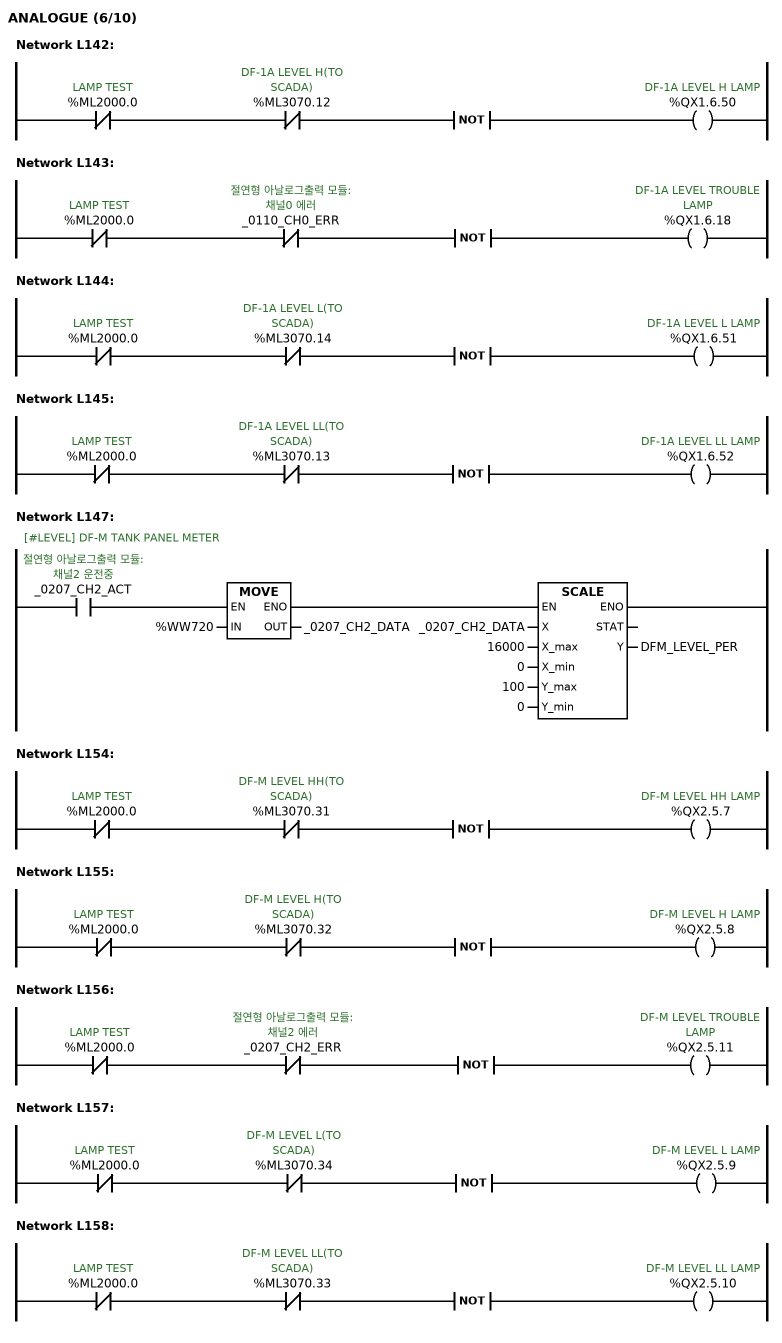
(* [picture p48: ANALOGUE rungs L142-L158] *)
(* Rung L142 *)
%QX1.6.50 := NOT (NOT %ML2000.0 AND NOT %ML3070.12);
(* Rung L143 *)
%QX1.6.18 := NOT (NOT %ML2000.0 AND NOT _0110_CH0_ERR);
(* Rung L144 *)
%QX1.6.51 := NOT (NOT %ML2000.0 AND NOT %ML3070.14);
(* Rung L145 *)
%QX1.6.52 := NOT (NOT %ML2000.0 AND NOT %ML3070.13);
(* [#LEVEL] DF-M TANK PANEL METER *)
(* Rung L147 *)
IF _0207_CH2_ACT THEN
    _0207_CH2_DATA := %WW720;
    SCALE(X := _0207_CH2_DATA, X_max := 16000, X_min := 0, Y_max := 100, Y_min := 0, Y => DFM_LEVEL_PER);
END_IF;
(* Rung L154 *)
%QX2.5.7 := NOT (NOT %ML2000.0 AND NOT %ML3070.31);
(* Rung L155 *)
%QX2.5.8 := NOT (NOT %ML2000.0 AND NOT %ML3070.32);
(* Rung L156 *)
%QX2.5.11 := NOT (NOT %ML2000.0 AND NOT _0207_CH2_ERR);
(* Rung L157 *)
%QX2.5.9 := NOT (NOT %ML2000.0 AND NOT %ML3070.34);
(* Rung L158 *)
%QX2.5.10 := NOT (NOT %ML2000.0 AND NOT %ML3070.33);

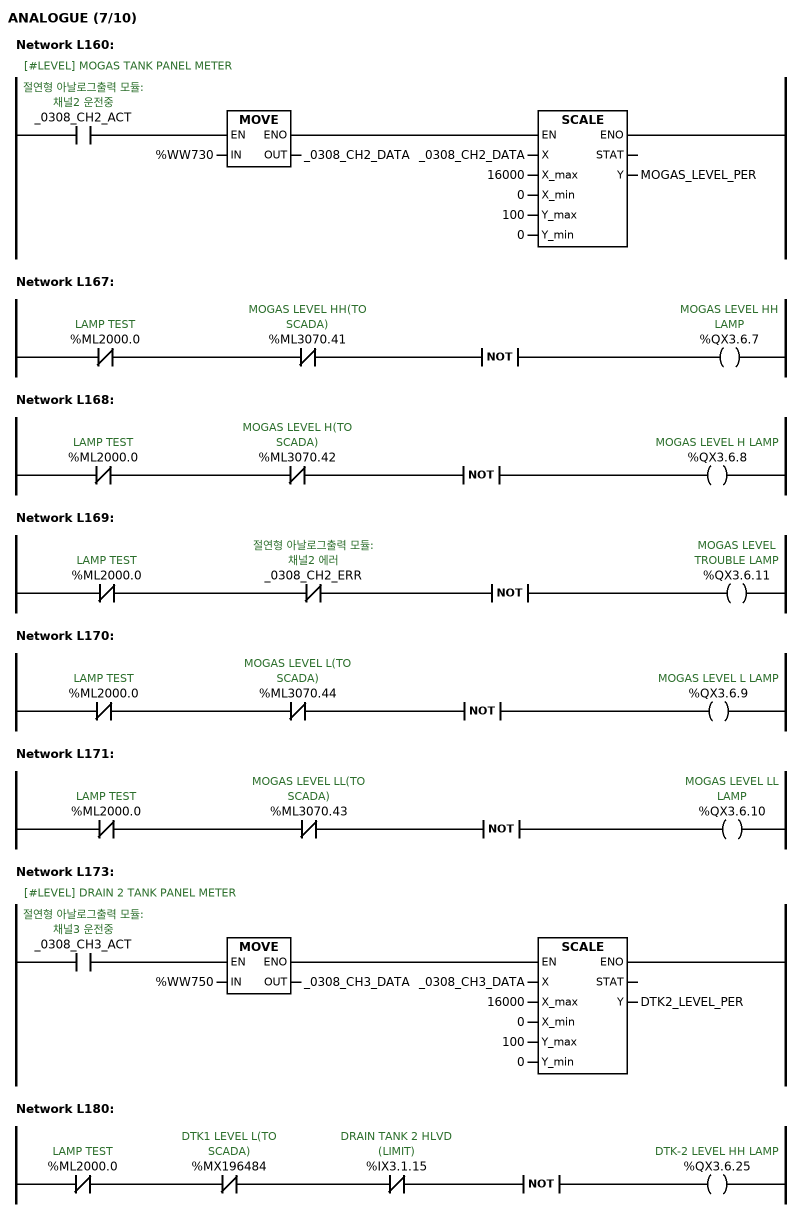
(* [#LEVEL] MOGAS TANK PANEL METER *)
(* Rung L160 *)
IF _0308_CH2_ACT THEN
    _0308_CH2_DATA := %WW730;
    SCALE(X := _0308_CH2_DATA, X_max := 16000, X_min := 0, Y_max := 100, Y_min := 0, Y => MOGAS_LEVEL_PER);
END_IF;
(* Rung L167 *)
%QX3.6.7 := NOT (NOT %ML2000.0 AND NOT %ML3070.41);
(* Rung L168 *)
%QX3.6.8 := NOT (NOT %ML2000.0 AND NOT %ML3070.42);
(* Rung L169 *)
%QX3.6.11 := NOT (NOT %ML2000.0 AND NOT _0308_CH2_ERR);
(* Rung L170 *)
%QX3.6.9 := NOT (NOT %ML2000.0 AND NOT %ML3070.44);
(* Rung L171 *)
%QX3.6.10 := NOT (NOT %ML2000.0 AND NOT %ML3070.43);
(* [#LEVEL] DRAIN 2 TANK PANEL METER *)
(* Rung L173 *)
IF _0308_CH3_ACT THEN
    _0308_CH3_DATA := %WW750;
    SCALE(X := _0308_CH3_DATA, X_max := 16000, X_min := 0, Y_max := 100, Y_min := 0, Y => DTK2_LEVEL_PER);
END_IF;
(* Rung L180 *)
%QX3.6.25 := NOT (NOT %ML2000.0 AND NOT %MX196484 AND NOT %IX3.1.15);

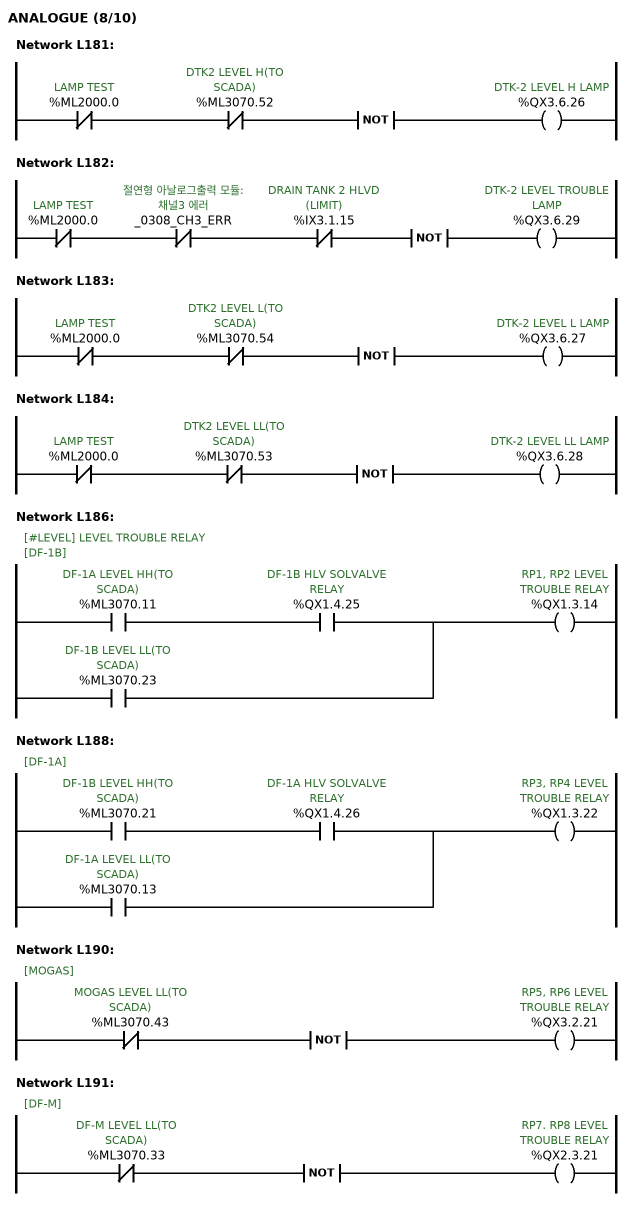
(* Rung L181 *)
%QX3.6.26 := NOT (NOT %ML2000.0 AND NOT %ML3070.52);
(* Rung L182 *)
%QX3.6.29 := NOT (NOT %ML2000.0 AND NOT _0308_CH3_ERR AND NOT %IX3.1.15);
(* Rung L183 *)
%QX3.6.27 := NOT (NOT %ML2000.0 AND NOT %ML3070.54);
(* Rung L184 *)
%QX3.6.28 := NOT (NOT %ML2000.0 AND NOT %ML3070.53);
(* [#LEVEL] LEVEL TROUBLE RELAY *)
(* Rung L186 *)
%QX1.3.14 := (%ML3070.11 AND %QX1.4.25) OR %ML3070.23;
(* [DF-1B] *)
(* Rung L188 *)
%QX1.3.22 := (%ML3070.21 AND %QX1.4.26) OR %ML3070.13;
(* [DF-1A] *)
(* Rung L190 *)
%QX3.2.21 := %ML3070.43;
(* [MOGAS] *)
(* Rung L191 *)
%QX2.3.21 := %ML3070.33;
(* [DF-M] *)

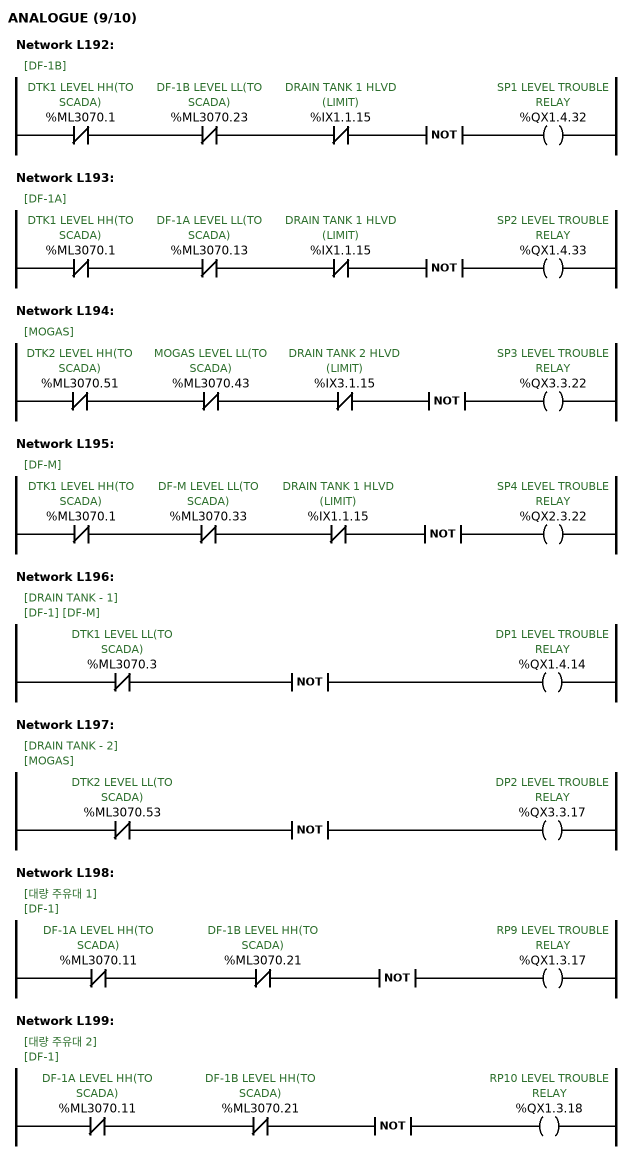
(* Rung L192 *)
%QX1.4.32 := NOT (NOT %ML3070.1 AND NOT %ML3070.23 AND NOT %IX1.1.15);
(* [DF-1B] *)
(* Rung L193 *)
%QX1.4.33 := NOT (NOT %ML3070.1 AND NOT %ML3070.13 AND NOT %IX1.1.15);
(* [DF-1A] *)
(* Rung L194 *)
%QX3.3.22 := NOT (NOT %ML3070.51 AND NOT %ML3070.43 AND NOT %IX3.1.15);
(* [MOGAS] *)
(* Rung L195 *)
%QX2.3.22 := NOT (NOT %ML3070.1 AND NOT %ML3070.33 AND NOT %IX1.1.15);
(* [DF-M] *)
(* Rung L196 *)
%QX1.4.14 := %ML3070.3;
(* [DRAIN TANK - 1] / [DF-1] [DF-M] *)
(* Rung L197 *)
%QX3.3.17 := %ML3070.53;
(* [DRAIN TANK - 2] / [MOGAS] *)
(* Rung L198 *)
%QX1.3.17 := NOT (NOT %ML3070.11 AND NOT %ML3070.21);
(* [대량 주유대 1] / [DF-1] *)
(* Rung L199 *)
%QX1.3.18 := NOT (NOT %ML3070.11 AND NOT %ML3070.21);
(* [대량 주유대 2] / [DF-1] *)

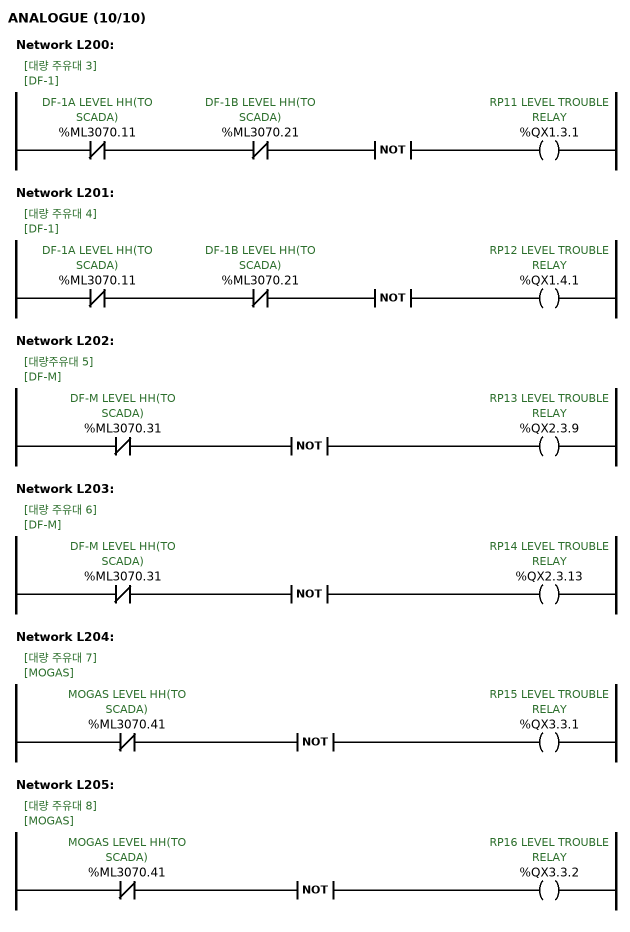
(* Rung L200 *)
%QX1.3.1 := NOT (NOT %ML3070.11 AND NOT %ML3070.21);
(* [대량 주유대 3] / [DF-1] *)
(* Rung L201 *)
%QX1.4.1 := NOT (NOT %ML3070.11 AND NOT %ML3070.21);
(* [대량 주유대 4] / [DF-1] *)
(* Rung L202 *)
%QX2.3.9 := %ML3070.31;
(* [대량주유대 5] / [DF-M] *)
(* Rung L203 *)
%QX2.3.13 := %ML3070.31;
(* [대량 주유대 6] / [DF-M] *)
(* Rung L204 *)
%QX3.3.1 := %ML3070.41;
(* [대량 주유대 7] / [MOGAS] *)
(* Rung L205 *)
%QX3.3.2 := %ML3070.41;
(* [대량 주유대 8] / [MOGAS] *)
END_PROGRAM

PROGRAM COMMUNICATION (* task: 스캔 프로그램 *)

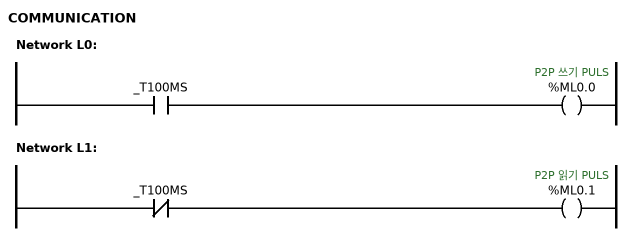
(* Rung L0 *)
%ML0.0 := _T100MS;
(* Rung L1 *)
%ML0.1 := NOT _T100MS;
END_PROGRAM

PROGRAM SCADA (* task: 스캔 프로그램 *)
VAR
    DFM_anyRun_SW : BOOL;
    MOGAS_anyRun_SW : BOOL;
END_VAR
VAR
    _t1 : BOOL;
    _t2 : BOOL;
END_VAR

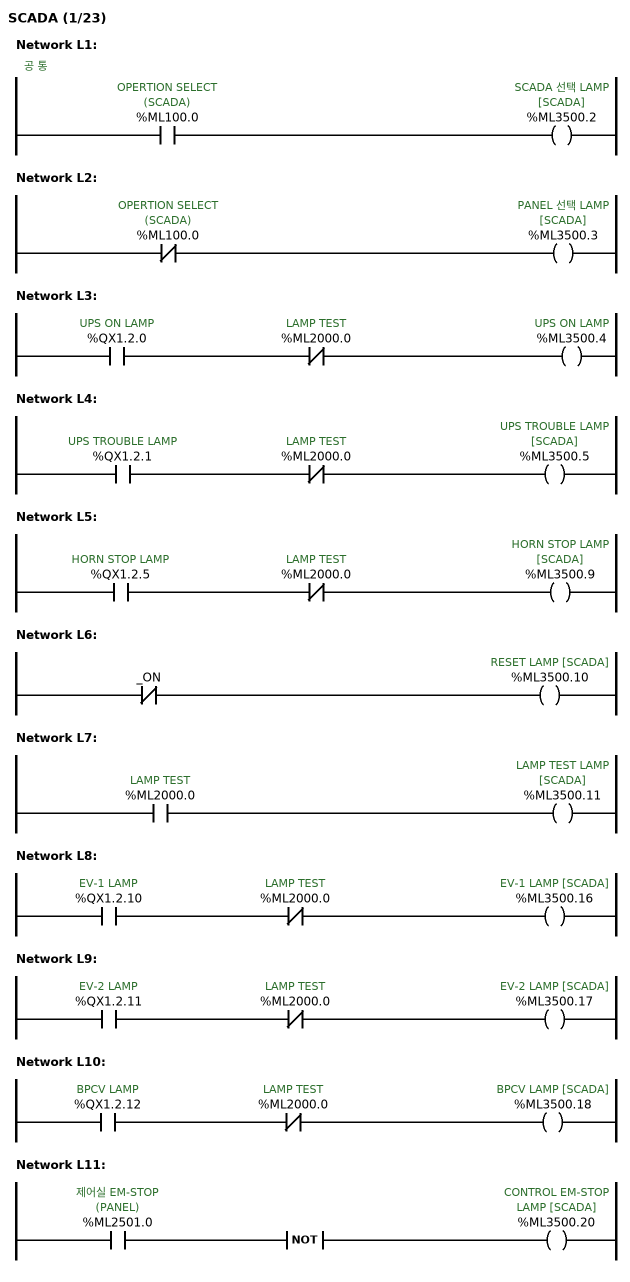
(* 공 통 *)
(* Rung L1 *)
%ML3500.2 := %ML100.0;
(* Rung L2 *)
%ML3500.3 := NOT %ML100.0;
(* Rung L3 *)
%ML3500.4 := %QX1.2.0 AND NOT %ML2000.0;
(* Rung L4 *)
%ML3500.5 := %QX1.2.1 AND NOT %ML2000.0;
(* Rung L5 *)
%ML3500.9 := %QX1.2.5 AND NOT %ML2000.0;
(* Rung L6 *)
%ML3500.10 := NOT _ON;
(* Rung L7 *)
%ML3500.11 := %ML2000.0;
(* Rung L8 *)
%ML3500.16 := %QX1.2.10 AND NOT %ML2000.0;
(* Rung L9 *)
%ML3500.17 := %QX1.2.11 AND NOT %ML2000.0;
(* Rung L10 *)
%ML3500.18 := %QX1.2.12 AND NOT %ML2000.0;
(* Rung L11 *)
%ML3500.20 := NOT %ML2501.0;

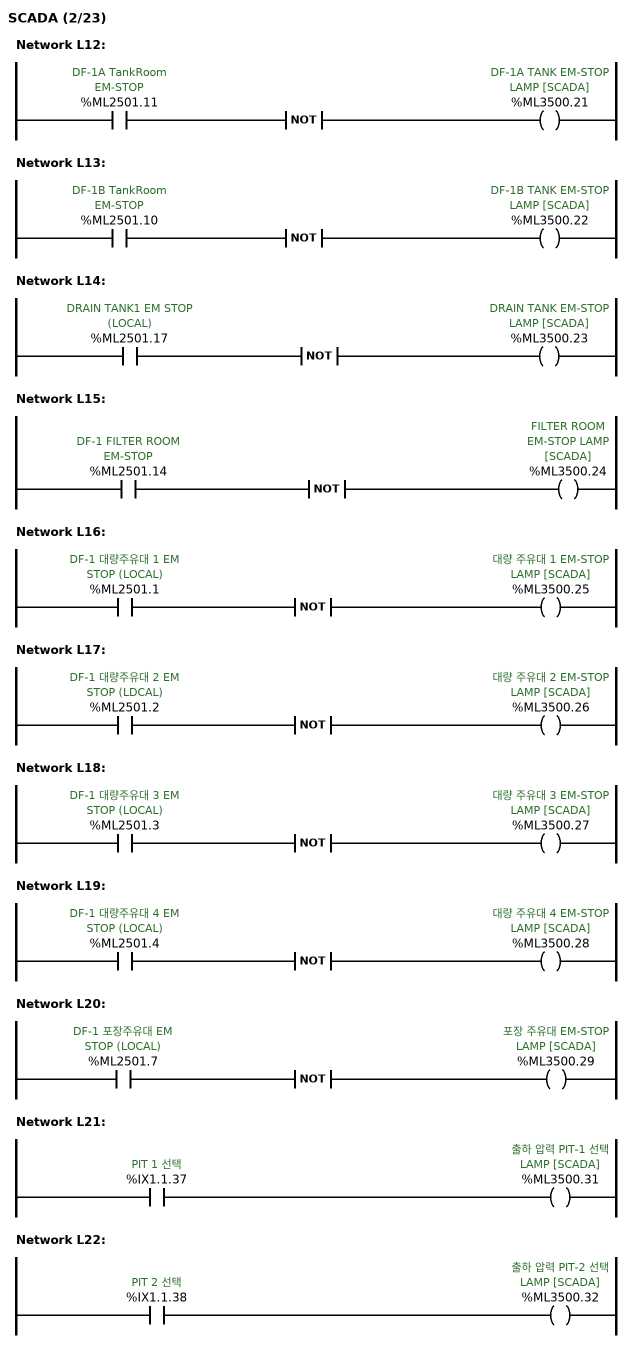
(* Rung L12 *)
%ML3500.21 := NOT %ML2501.11;
(* Rung L13 *)
%ML3500.22 := NOT %ML2501.10;
(* Rung L14 *)
%ML3500.23 := NOT %ML2501.17;
(* Rung L15 *)
%ML3500.24 := NOT %ML2501.14;
(* Rung L16 *)
%ML3500.25 := NOT %ML2501.1;
(* Rung L17 *)
%ML3500.26 := NOT %ML2501.2;
(* Rung L18 *)
%ML3500.27 := NOT %ML2501.3;
(* Rung L19 *)
%ML3500.28 := NOT %ML2501.4;
(* Rung L20 *)
%ML3500.29 := NOT %ML2501.7;
(* Rung L21 *)
%ML3500.31 := %IX1.1.37;
(* Rung L22 *)
%ML3500.32 := %IX1.1.38;

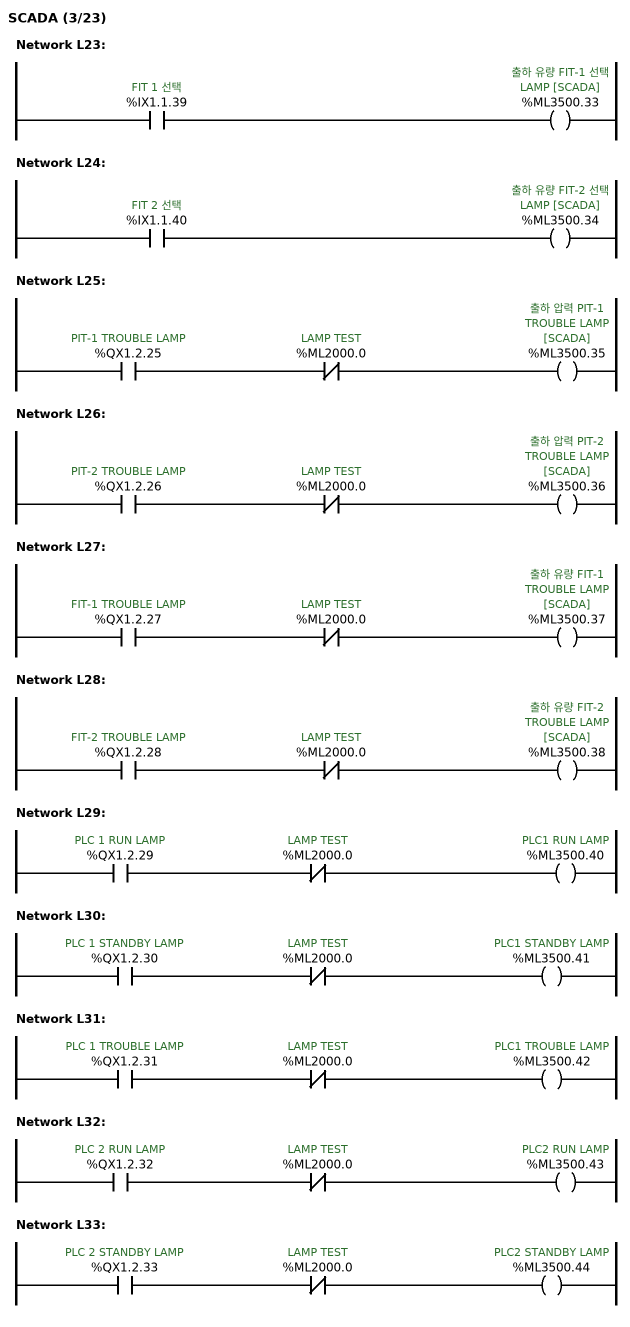
(* Rung L23 *)
%ML3500.33 := %IX1.1.39;
(* Rung L24 *)
%ML3500.34 := %IX1.1.40;
(* Rung L25 *)
%ML3500.35 := %QX1.2.25 AND NOT %ML2000.0;
(* Rung L26 *)
%ML3500.36 := %QX1.2.26 AND NOT %ML2000.0;
(* Rung L27 *)
%ML3500.37 := %QX1.2.27 AND NOT %ML2000.0;
(* Rung L28 *)
%ML3500.38 := %QX1.2.28 AND NOT %ML2000.0;
(* Rung L29 *)
%ML3500.40 := %QX1.2.29 AND NOT %ML2000.0;
(* Rung L30 *)
%ML3500.41 := %QX1.2.30 AND NOT %ML2000.0;
(* Rung L31 *)
%ML3500.42 := %QX1.2.31 AND NOT %ML2000.0;
(* Rung L32 *)
%ML3500.43 := %QX1.2.32 AND NOT %ML2000.0;
(* Rung L33 *)
%ML3500.44 := %QX1.2.33 AND NOT %ML2000.0;

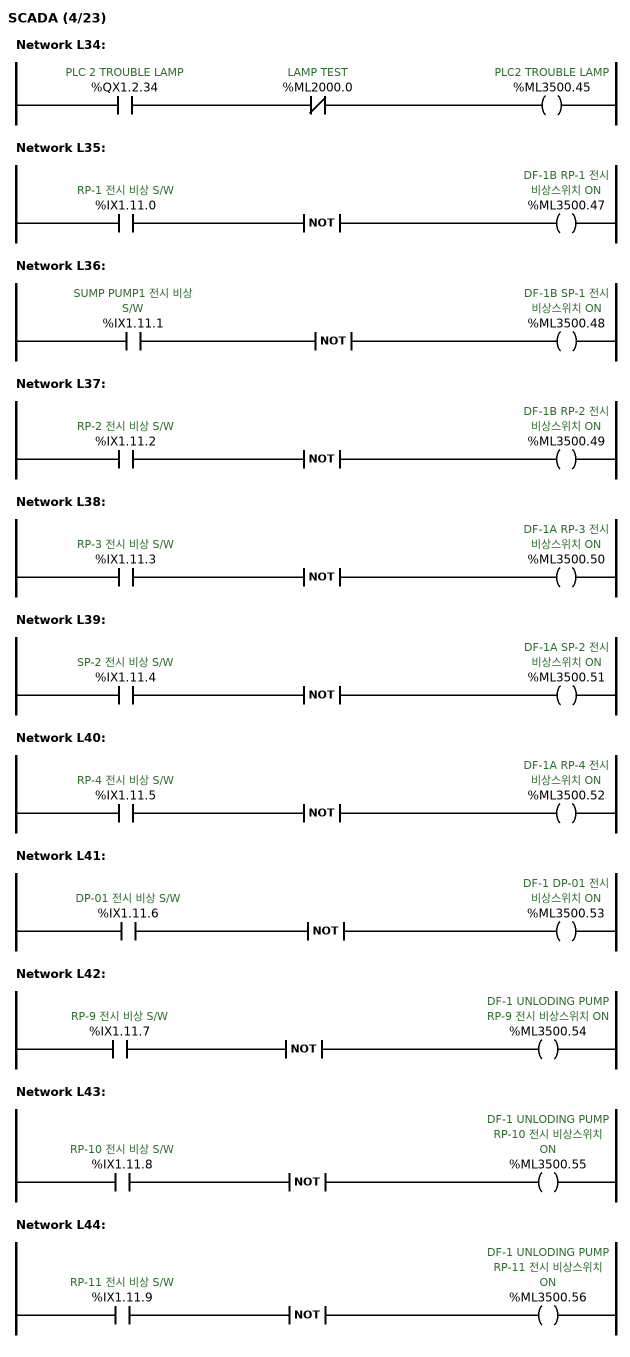
(* Rung L34 *)
%ML3500.45 := %QX1.2.34 AND NOT %ML2000.0;
(* Rung L35 *)
%ML3500.47 := NOT %IX1.11.0;
(* Rung L36 *)
%ML3500.48 := NOT %IX1.11.1;
(* Rung L37 *)
%ML3500.49 := NOT %IX1.11.2;
(* Rung L38 *)
%ML3500.50 := NOT %IX1.11.3;
(* Rung L39 *)
%ML3500.51 := NOT %IX1.11.4;
(* Rung L40 *)
%ML3500.52 := NOT %IX1.11.5;
(* Rung L41 *)
%ML3500.53 := NOT %IX1.11.6;
(* Rung L42 *)
%ML3500.54 := NOT %IX1.11.7;
(* Rung L43 *)
%ML3500.55 := NOT %IX1.11.8;
(* Rung L44 *)
%ML3500.56 := NOT %IX1.11.9;

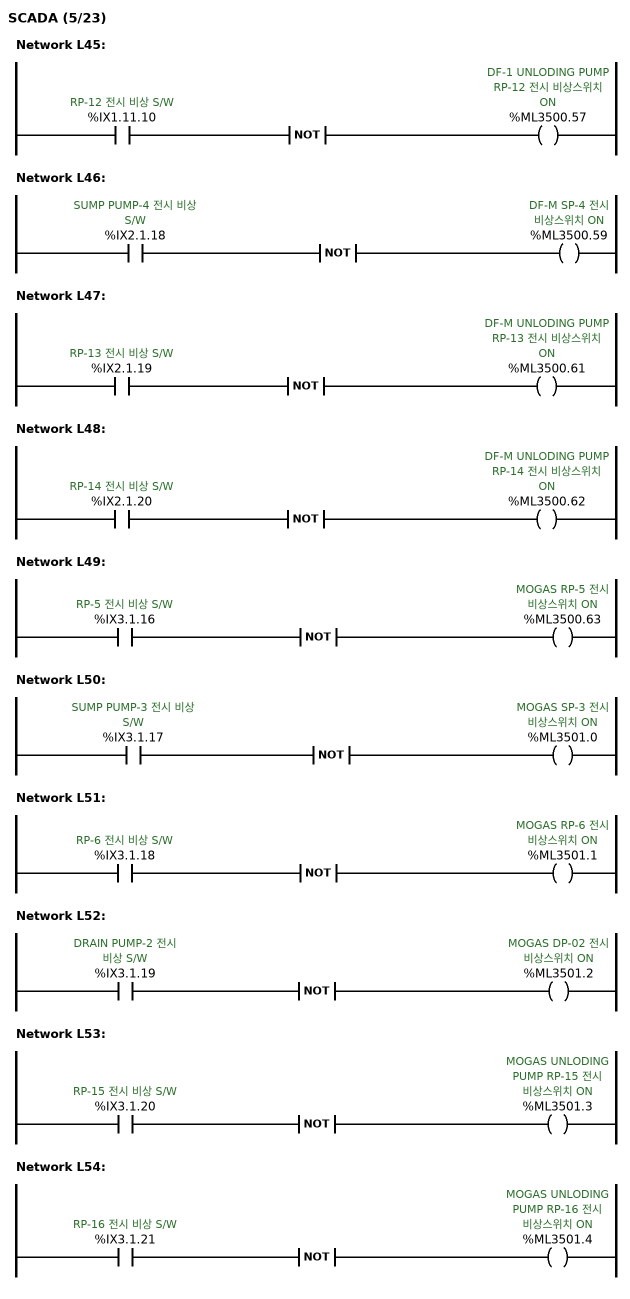
(* Rung L45 *)
%ML3500.57 := NOT %IX1.11.10;
(* Rung L46 *)
%ML3500.59 := NOT %IX2.1.18;
(* Rung L47 *)
%ML3500.61 := NOT %IX2.1.19;
(* Rung L48 *)
%ML3500.62 := NOT %IX2.1.20;
(* Rung L49 *)
%ML3500.63 := NOT %IX3.1.16;
(* Rung L50 *)
%ML3501.0 := NOT %IX3.1.17;
(* Rung L51 *)
%ML3501.1 := NOT %IX3.1.18;
(* Rung L52 *)
%ML3501.2 := NOT %IX3.1.19;
(* Rung L53 *)
%ML3501.3 := NOT %IX3.1.20;
(* Rung L54 *)
%ML3501.4 := NOT %IX3.1.21;

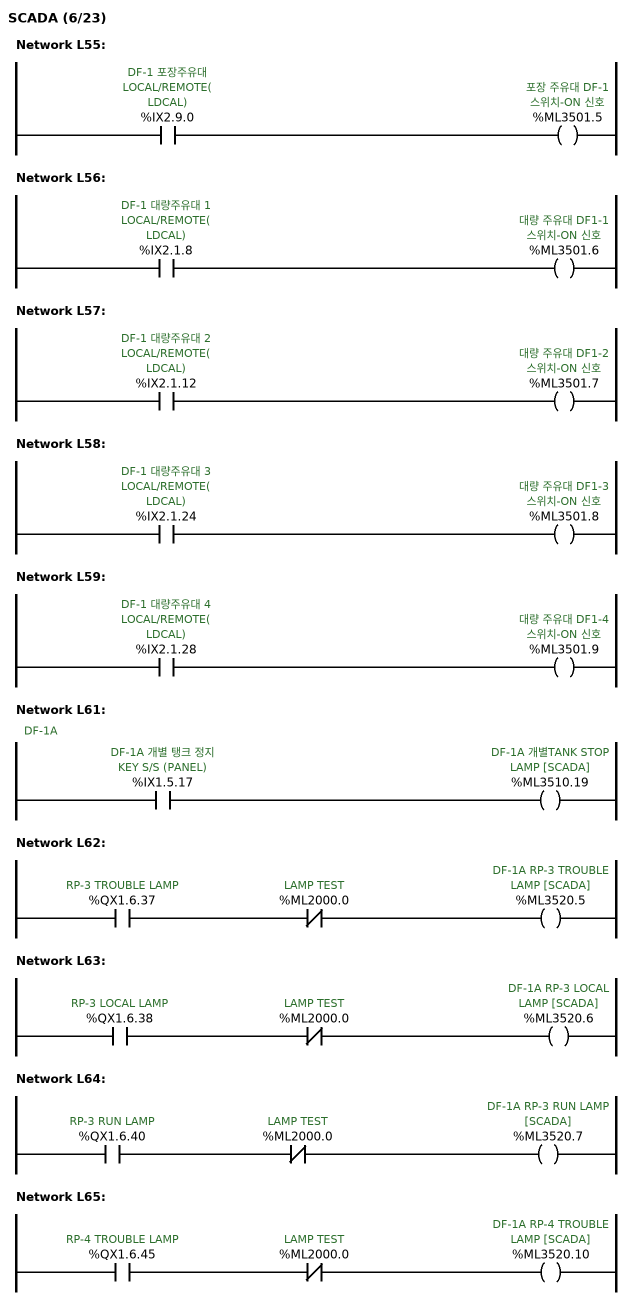
(* Rung L55 *)
%ML3501.5 := %IX2.9.0;
(* Rung L56 *)
%ML3501.6 := %IX2.1.8;
(* Rung L57 *)
%ML3501.7 := %IX2.1.12;
(* Rung L58 *)
%ML3501.8 := %IX2.1.24;
(* Rung L59 *)
%ML3501.9 := %IX2.1.28;
(* DF-1A *)
(* Rung L61 *)
%ML3510.19 := %IX1.5.17;
(* Rung L62 *)
%ML3520.5 := %QX1.6.37 AND NOT %ML2000.0;
(* Rung L63 *)
%ML3520.6 := %QX1.6.38 AND NOT %ML2000.0;
(* Rung L64 *)
%ML3520.7 := %QX1.6.40 AND NOT %ML2000.0;
(* Rung L65 *)
%ML3520.10 := %QX1.6.45 AND NOT %ML2000.0;

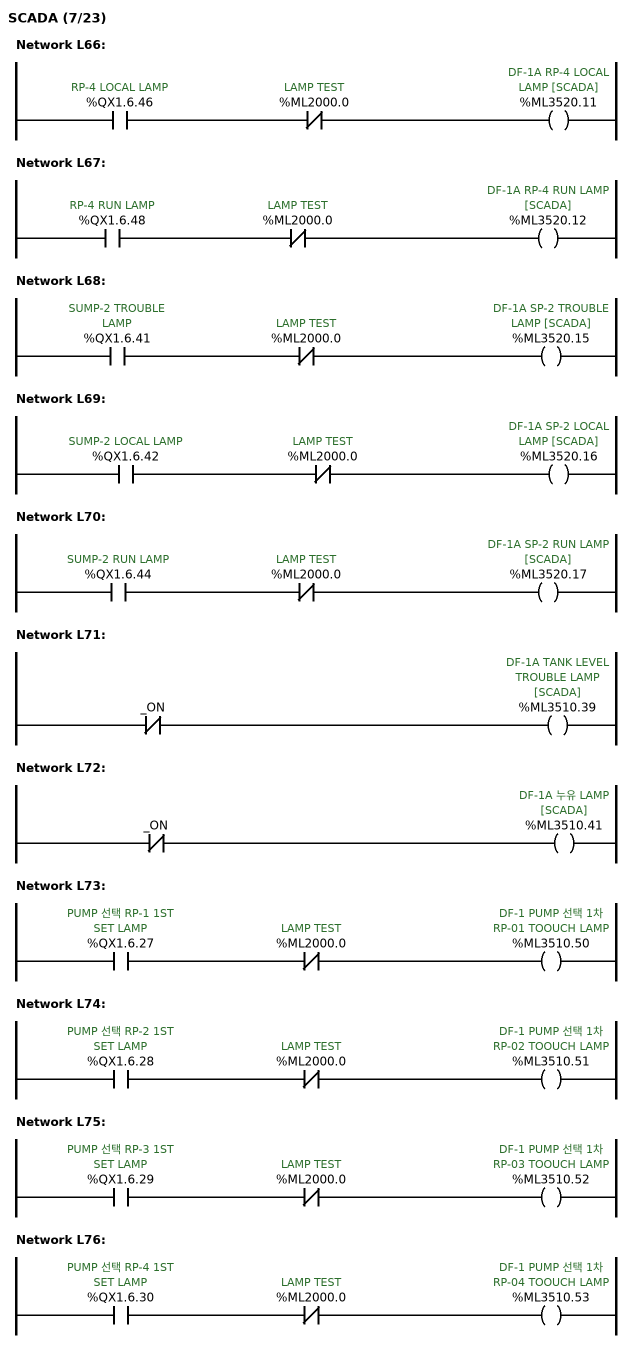
(* Rung L66 *)
%ML3520.11 := %QX1.6.46 AND NOT %ML2000.0;
(* Rung L67 *)
%ML3520.12 := %QX1.6.48 AND NOT %ML2000.0;
(* Rung L68 *)
%ML3520.15 := %QX1.6.41 AND NOT %ML2000.0;
(* Rung L69 *)
%ML3520.16 := %QX1.6.42 AND NOT %ML2000.0;
(* Rung L70 *)
%ML3520.17 := %QX1.6.44 AND NOT %ML2000.0;
(* Rung L71 *)
%ML3510.39 := NOT _ON;
(* Rung L72 *)
%ML3510.41 := NOT _ON;
(* Rung L73 *)
%ML3510.50 := %QX1.6.27 AND NOT %ML2000.0;
(* Rung L74 *)
%ML3510.51 := %QX1.6.28 AND NOT %ML2000.0;
(* Rung L75 *)
%ML3510.52 := %QX1.6.29 AND NOT %ML2000.0;
(* Rung L76 *)
%ML3510.53 := %QX1.6.30 AND NOT %ML2000.0;

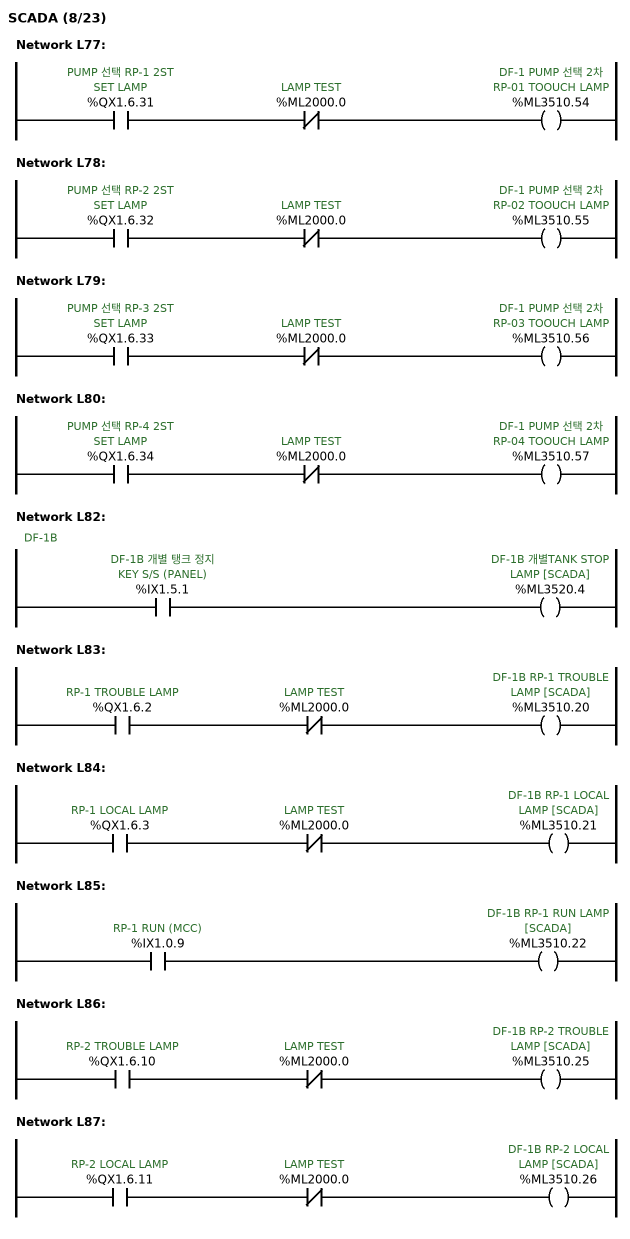
(* Rung L77 *)
%ML3510.54 := %QX1.6.31 AND NOT %ML2000.0;
(* Rung L78 *)
%ML3510.55 := %QX1.6.32 AND NOT %ML2000.0;
(* Rung L79 *)
%ML3510.56 := %QX1.6.33 AND NOT %ML2000.0;
(* Rung L80 *)
%ML3510.57 := %QX1.6.34 AND NOT %ML2000.0;
(* DF-1B *)
(* Rung L82 *)
%ML3520.4 := %IX1.5.1;
(* Rung L83 *)
%ML3510.20 := %QX1.6.2 AND NOT %ML2000.0;
(* Rung L84 *)
%ML3510.21 := %QX1.6.3 AND NOT %ML2000.0;
(* Rung L85 *)
%ML3510.22 := %IX1.0.9;
(* Rung L86 *)
%ML3510.25 := %QX1.6.10 AND NOT %ML2000.0;
(* Rung L87 *)
%ML3510.26 := %QX1.6.11 AND NOT %ML2000.0;

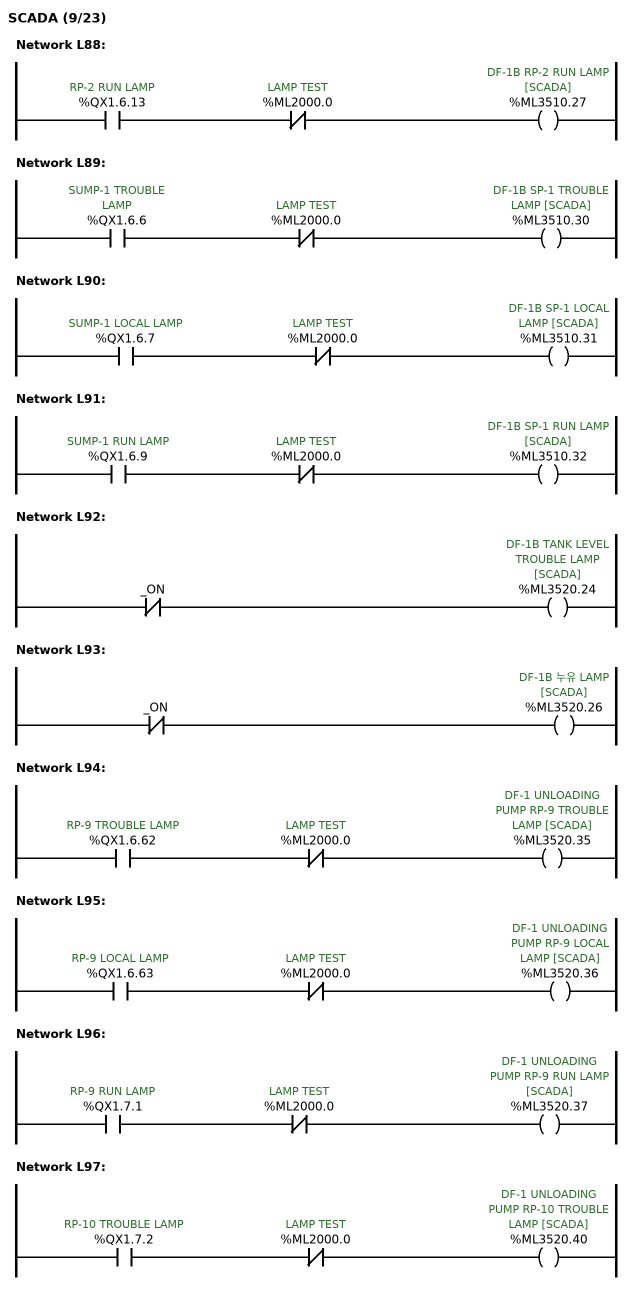
(* Rung L88 *)
%ML3510.27 := %QX1.6.13 AND NOT %ML2000.0;
(* Rung L89 *)
%ML3510.30 := %QX1.6.6 AND NOT %ML2000.0;
(* Rung L90 *)
%ML3510.31 := %QX1.6.7 AND NOT %ML2000.0;
(* Rung L91 *)
%ML3510.32 := %QX1.6.9 AND NOT %ML2000.0;
(* Rung L92 *)
%ML3520.24 := NOT _ON;
(* Rung L93 *)
%ML3520.26 := NOT _ON;
(* Rung L94 *)
%ML3520.35 := %QX1.6.62 AND NOT %ML2000.0;
(* Rung L95 *)
%ML3520.36 := %QX1.6.63 AND NOT %ML2000.0;
(* Rung L96 *)
%ML3520.37 := %QX1.7.1 AND NOT %ML2000.0;
(* Rung L97 *)
%ML3520.40 := %QX1.7.2 AND NOT %ML2000.0;

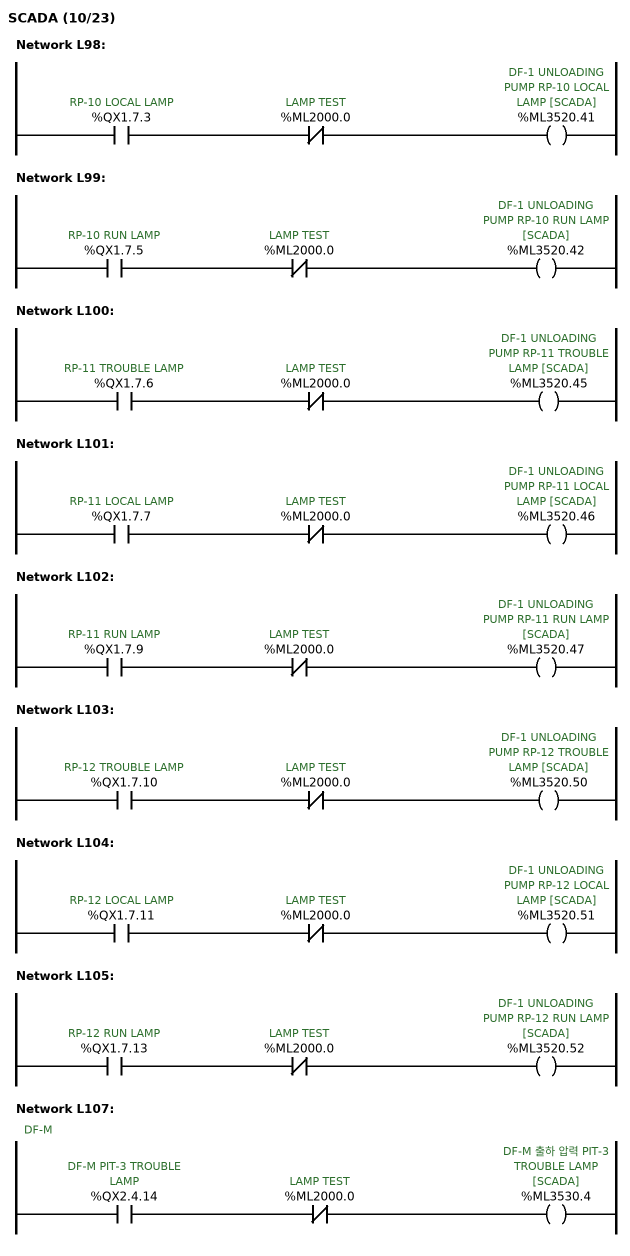
(* Rung L98 *)
%ML3520.41 := %QX1.7.3 AND NOT %ML2000.0;
(* Rung L99 *)
%ML3520.42 := %QX1.7.5 AND NOT %ML2000.0;
(* Rung L100 *)
%ML3520.45 := %QX1.7.6 AND NOT %ML2000.0;
(* Rung L101 *)
%ML3520.46 := %QX1.7.7 AND NOT %ML2000.0;
(* Rung L102 *)
%ML3520.47 := %QX1.7.9 AND NOT %ML2000.0;
(* Rung L103 *)
%ML3520.50 := %QX1.7.10 AND NOT %ML2000.0;
(* Rung L104 *)
%ML3520.51 := %QX1.7.11 AND NOT %ML2000.0;
(* Rung L105 *)
%ML3520.52 := %QX1.7.13 AND NOT %ML2000.0;
(* DF-M *)
(* Rung L107 *)
%ML3530.4 := %QX2.4.14 AND NOT %ML2000.0;

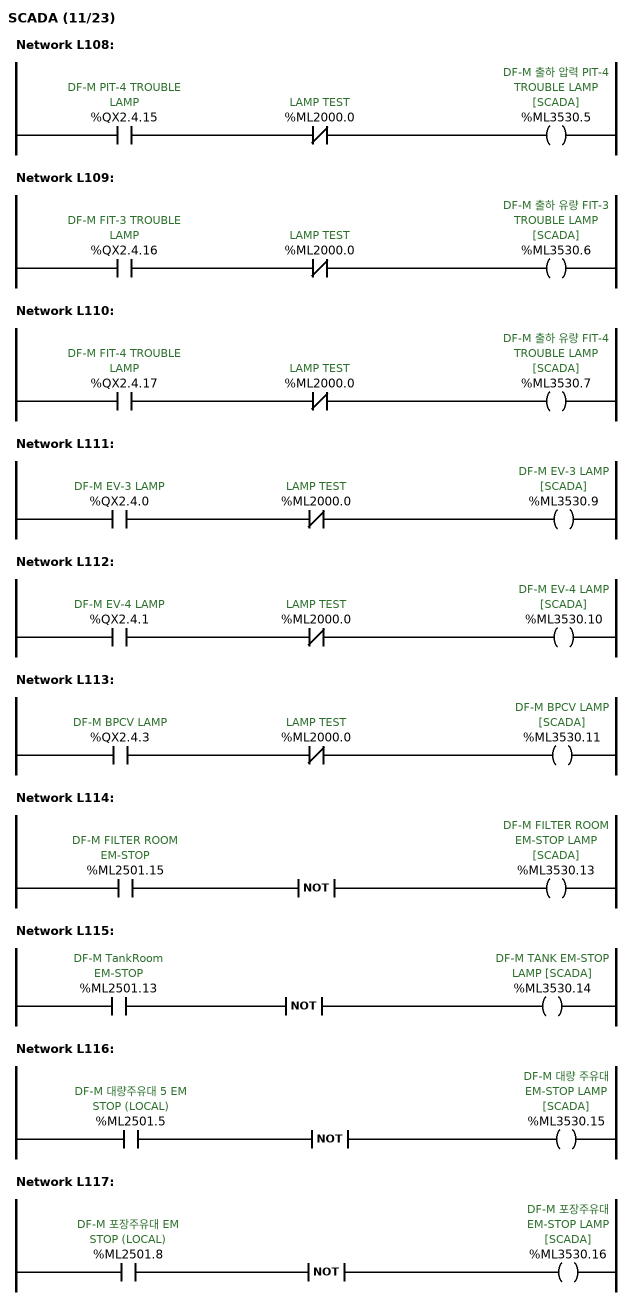
(* Rung L108 *)
%ML3530.5 := %QX2.4.15 AND NOT %ML2000.0;
(* Rung L109 *)
%ML3530.6 := %QX2.4.16 AND NOT %ML2000.0;
(* Rung L110 *)
%ML3530.7 := %QX2.4.17 AND NOT %ML2000.0;
(* Rung L111 *)
%ML3530.9 := %QX2.4.0 AND NOT %ML2000.0;
(* Rung L112 *)
%ML3530.10 := %QX2.4.1 AND NOT %ML2000.0;
(* Rung L113 *)
%ML3530.11 := %QX2.4.3 AND NOT %ML2000.0;
(* Rung L114 *)
%ML3530.13 := NOT %ML2501.15;
(* Rung L115 *)
%ML3530.14 := NOT %ML2501.13;
(* Rung L116 *)
%ML3530.15 := NOT %ML2501.5;
(* Rung L117 *)
%ML3530.16 := NOT %ML2501.8;

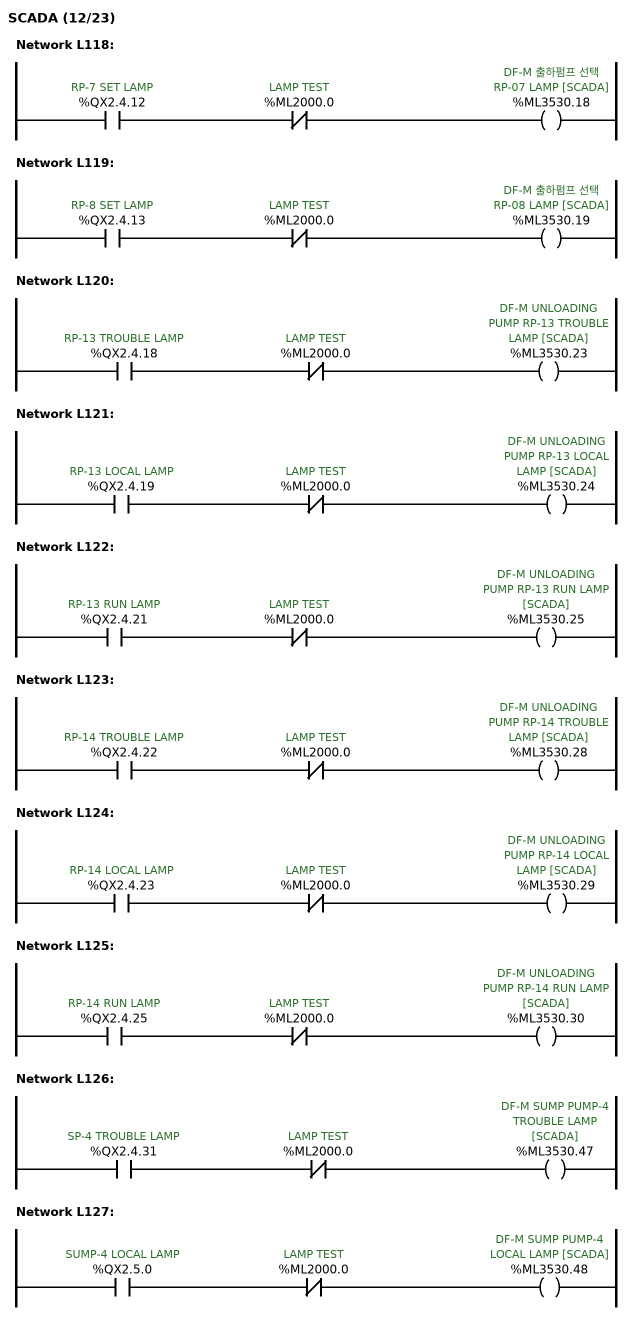
(* Rung L118 *)
%ML3530.18 := %QX2.4.12 AND NOT %ML2000.0;
(* Rung L119 *)
%ML3530.19 := %QX2.4.13 AND NOT %ML2000.0;
(* Rung L120 *)
%ML3530.23 := %QX2.4.18 AND NOT %ML2000.0;
(* Rung L121 *)
%ML3530.24 := %QX2.4.19 AND NOT %ML2000.0;
(* Rung L122 *)
%ML3530.25 := %QX2.4.21 AND NOT %ML2000.0;
(* Rung L123 *)
%ML3530.28 := %QX2.4.22 AND NOT %ML2000.0;
(* Rung L124 *)
%ML3530.29 := %QX2.4.23 AND NOT %ML2000.0;
(* Rung L125 *)
%ML3530.30 := %QX2.4.25 AND NOT %ML2000.0;
(* Rung L126 *)
%ML3530.47 := %QX2.4.31 AND NOT %ML2000.0;
(* Rung L127 *)
%ML3530.48 := %QX2.5.0 AND NOT %ML2000.0;

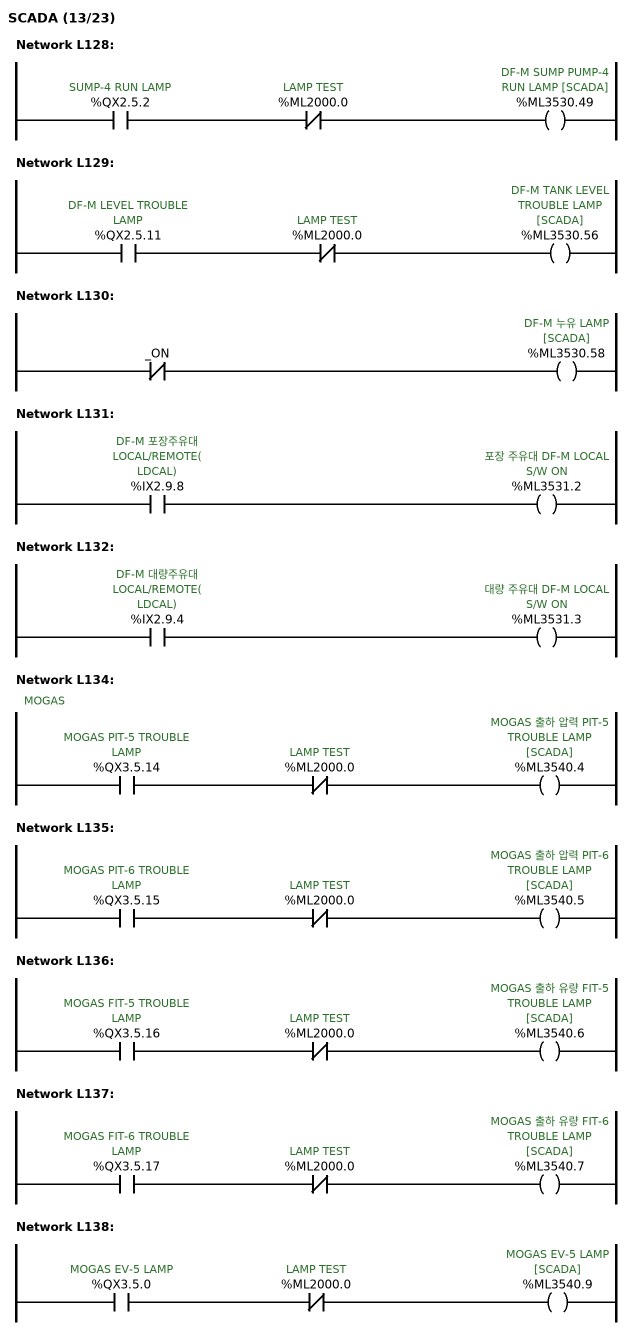
(* Rung L128 *)
%ML3530.49 := %QX2.5.2 AND NOT %ML2000.0;
(* Rung L129 *)
%ML3530.56 := %QX2.5.11 AND NOT %ML2000.0;
(* Rung L130 *)
%ML3530.58 := NOT _ON;
(* Rung L131 *)
%ML3531.2 := %IX2.9.8;
(* Rung L132 *)
%ML3531.3 := %IX2.9.4;
(* MOGAS *)
(* Rung L134 *)
%ML3540.4 := %QX3.5.14 AND NOT %ML2000.0;
(* Rung L135 *)
%ML3540.5 := %QX3.5.15 AND NOT %ML2000.0;
(* Rung L136 *)
%ML3540.6 := %QX3.5.16 AND NOT %ML2000.0;
(* Rung L137 *)
%ML3540.7 := %QX3.5.17 AND NOT %ML2000.0;
(* Rung L138 *)
%ML3540.9 := %QX3.5.0 AND NOT %ML2000.0;

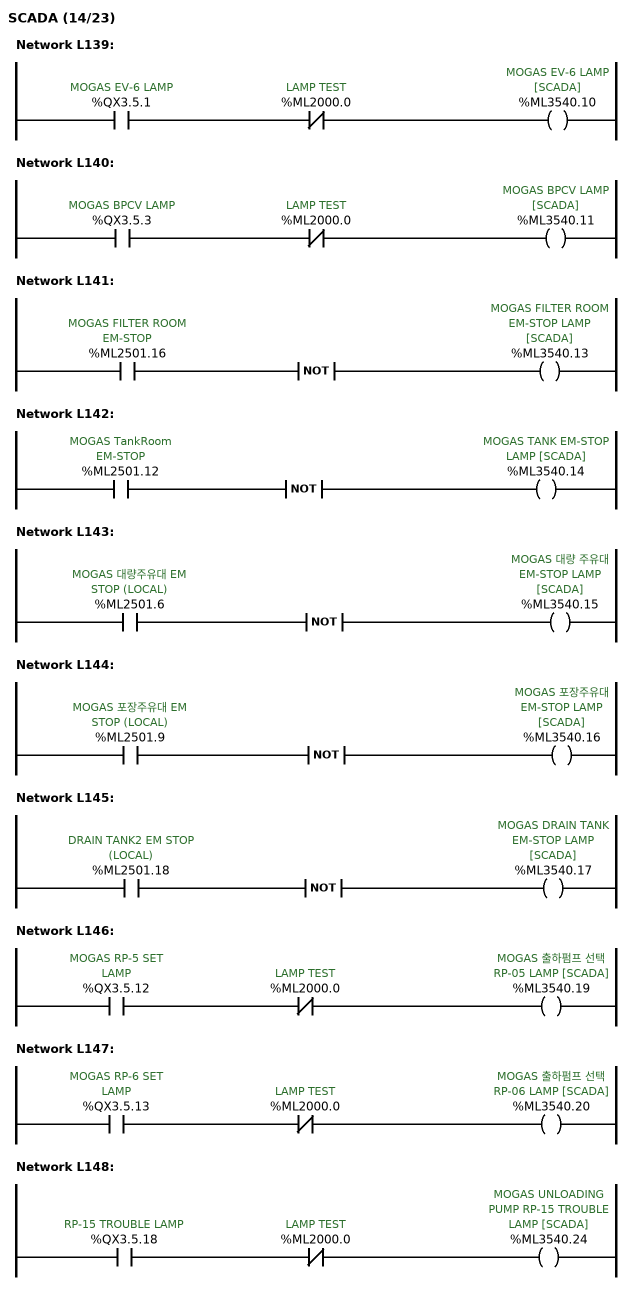
(* Rung L139 *)
%ML3540.10 := %QX3.5.1 AND NOT %ML2000.0;
(* Rung L140 *)
%ML3540.11 := %QX3.5.3 AND NOT %ML2000.0;
(* Rung L141 *)
%ML3540.13 := NOT %ML2501.16;
(* Rung L142 *)
%ML3540.14 := NOT %ML2501.12;
(* Rung L143 *)
%ML3540.15 := NOT %ML2501.6;
(* Rung L144 *)
%ML3540.16 := NOT %ML2501.9;
(* Rung L145 *)
%ML3540.17 := NOT %ML2501.18;
(* Rung L146 *)
%ML3540.19 := %QX3.5.12 AND NOT %ML2000.0;
(* Rung L147 *)
%ML3540.20 := %QX3.5.13 AND NOT %ML2000.0;
(* Rung L148 *)
%ML3540.24 := %QX3.5.18 AND NOT %ML2000.0;

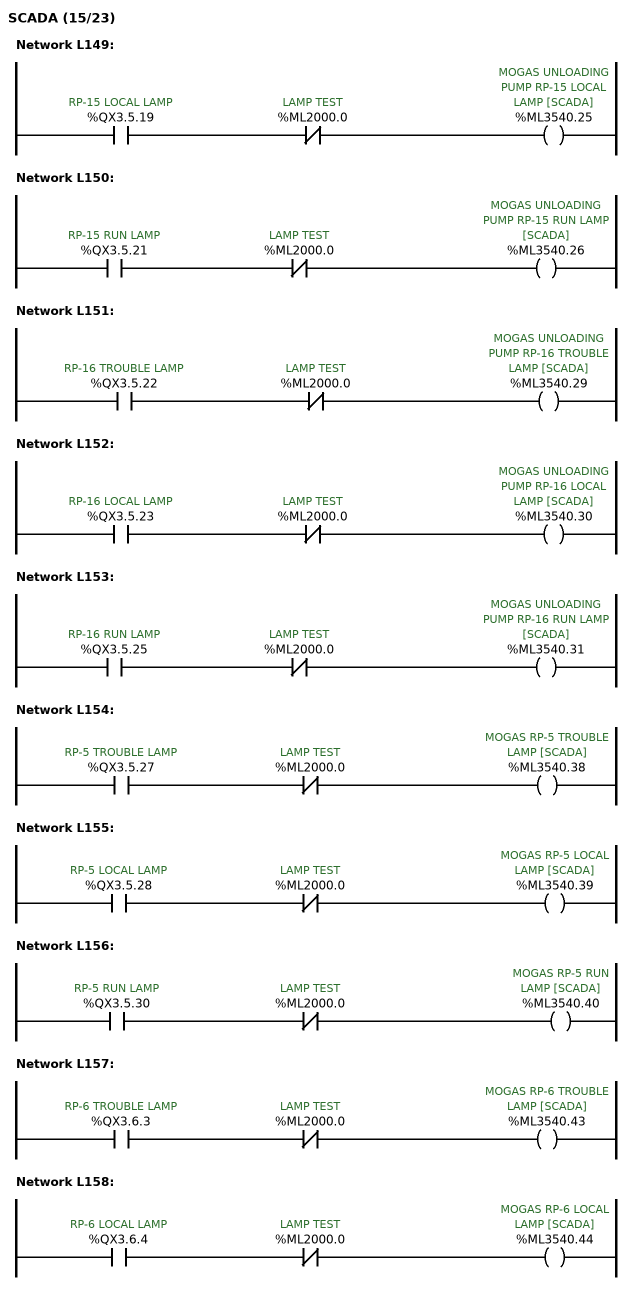
(* Rung L149 *)
%ML3540.25 := %QX3.5.19 AND NOT %ML2000.0;
(* Rung L150 *)
%ML3540.26 := %QX3.5.21 AND NOT %ML2000.0;
(* Rung L151 *)
%ML3540.29 := %QX3.5.22 AND NOT %ML2000.0;
(* Rung L152 *)
%ML3540.30 := %QX3.5.23 AND NOT %ML2000.0;
(* Rung L153 *)
%ML3540.31 := %QX3.5.25 AND NOT %ML2000.0;
(* Rung L154 *)
%ML3540.38 := %QX3.5.27 AND NOT %ML2000.0;
(* Rung L155 *)
%ML3540.39 := %QX3.5.28 AND NOT %ML2000.0;
(* Rung L156 *)
%ML3540.40 := %QX3.5.30 AND NOT %ML2000.0;
(* Rung L157 *)
%ML3540.43 := %QX3.6.3 AND NOT %ML2000.0;
(* Rung L158 *)
%ML3540.44 := %QX3.6.4 AND NOT %ML2000.0;

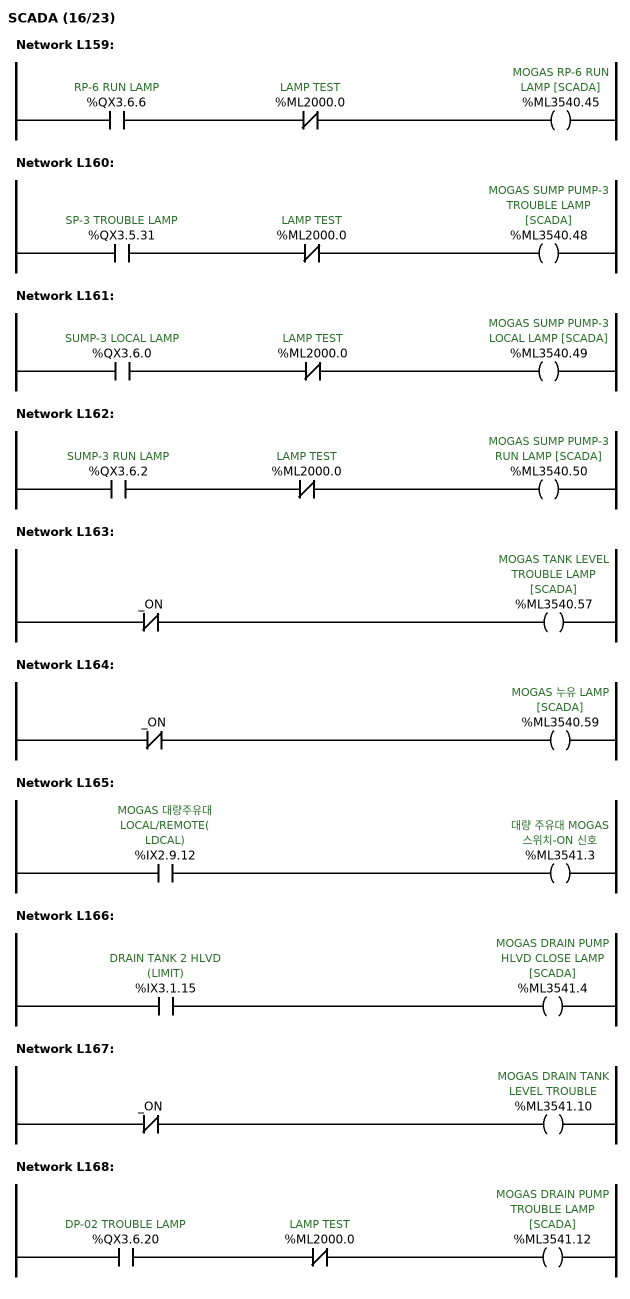
(* Rung L159 *)
%ML3540.45 := %QX3.6.6 AND NOT %ML2000.0;
(* Rung L160 *)
%ML3540.48 := %QX3.5.31 AND NOT %ML2000.0;
(* Rung L161 *)
%ML3540.49 := %QX3.6.0 AND NOT %ML2000.0;
(* Rung L162 *)
%ML3540.50 := %QX3.6.2 AND NOT %ML2000.0;
(* Rung L163 *)
%ML3540.57 := NOT _ON;
(* Rung L164 *)
%ML3540.59 := NOT _ON;
(* Rung L165 *)
%ML3541.3 := %IX2.9.12;
(* Rung L166 *)
%ML3541.4 := %IX3.1.15;
(* Rung L167 *)
%ML3541.10 := NOT _ON;
(* Rung L168 *)
%ML3541.12 := %QX3.6.20 AND NOT %ML2000.0;

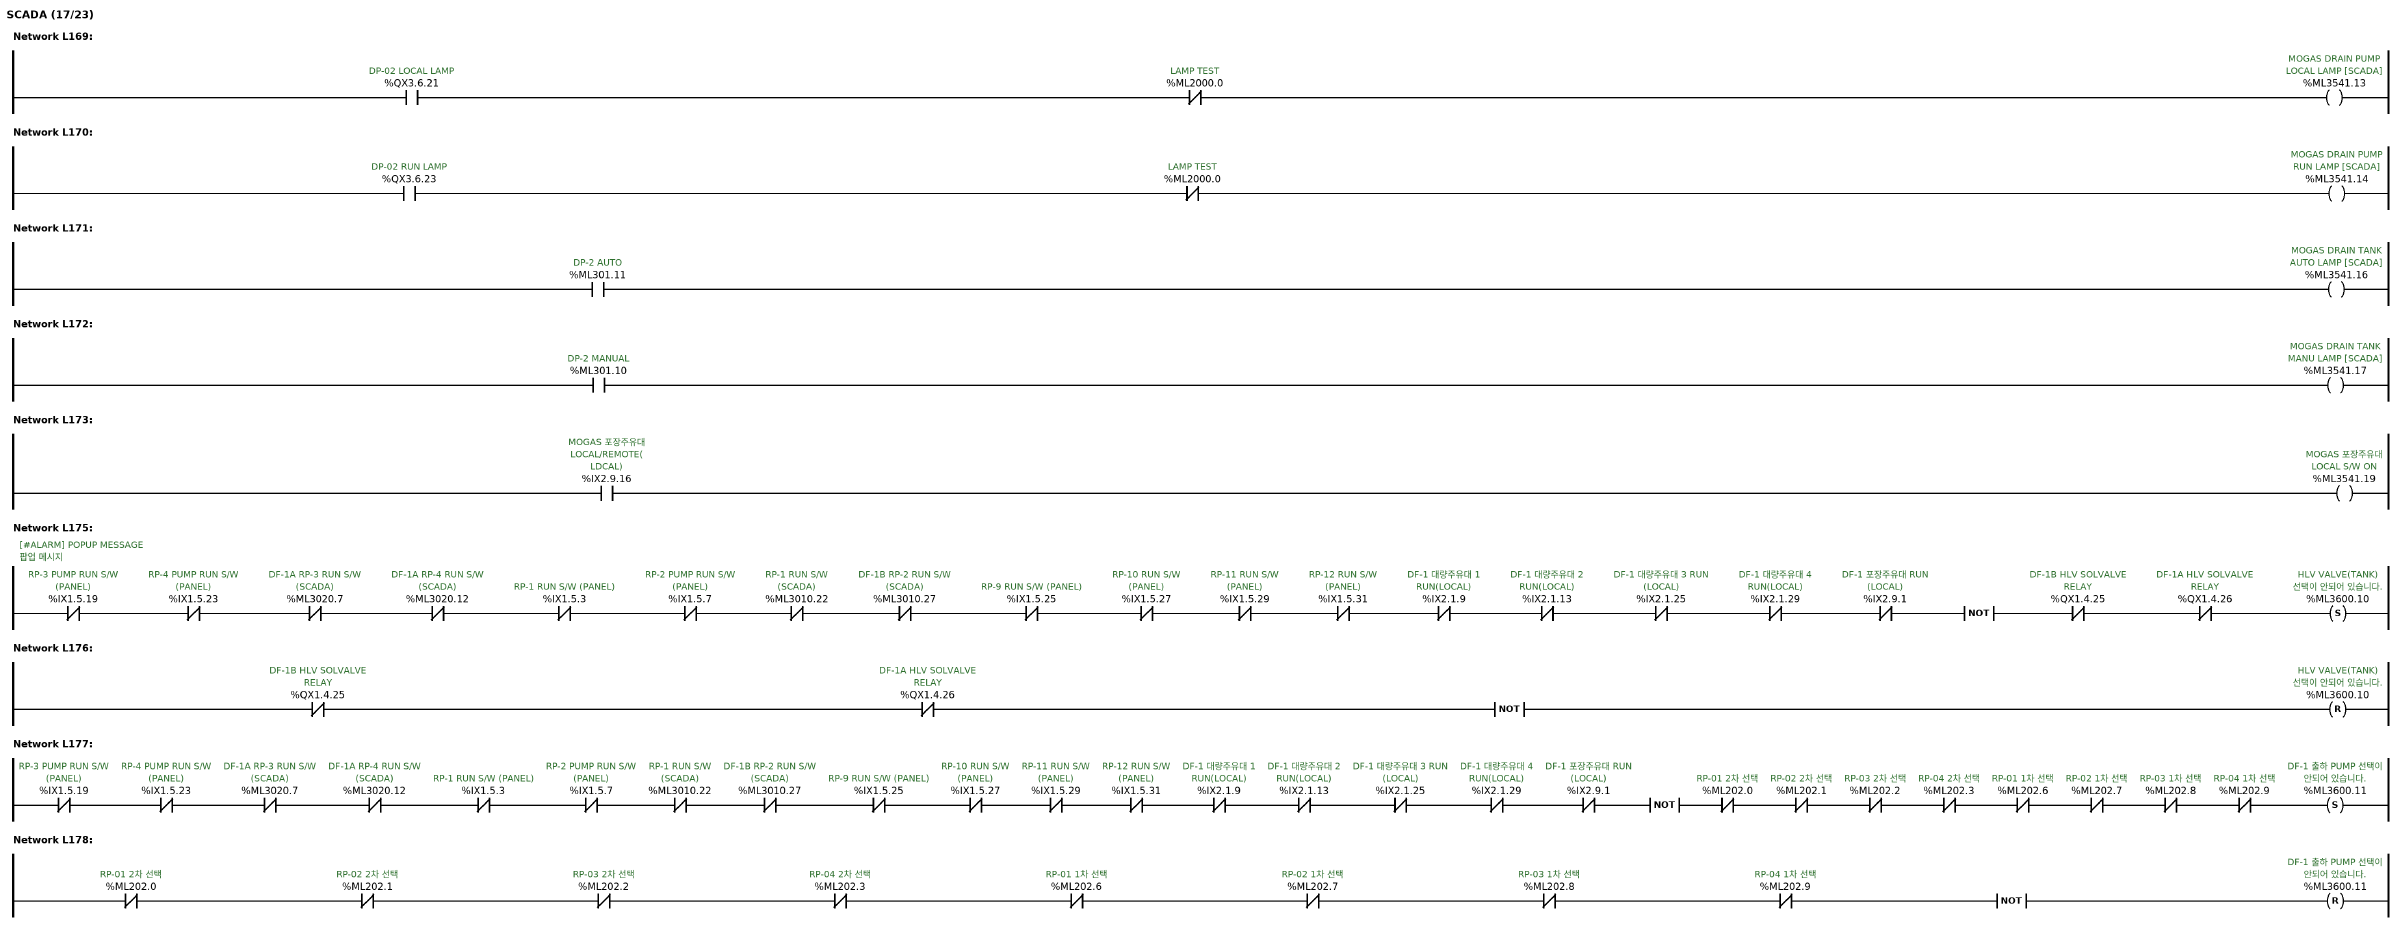
(* Rung L169 *)
%ML3541.13 := %QX3.6.21 AND NOT %ML2000.0;
(* Rung L170 *)
%ML3541.14 := %QX3.6.23 AND NOT %ML2000.0;
(* Rung L171 *)
%ML3541.16 := %ML301.11;
(* Rung L172 *)
%ML3541.17 := %ML301.10;
(* Rung L173 *)
%ML3541.19 := %IX2.9.16;
(* [#ALARM] POPUP MESSAGE *)
(* Rung L175 *)
IF NOT (NOT %IX1.5.19 AND NOT %IX1.5.23 AND NOT %ML3020.7 AND NOT %ML3020.12 AND NOT %IX1.5.3 AND NOT %IX1.5.7 AND NOT %ML3010.22 AND NOT %ML3010.27 AND NOT %IX1.5.25 AND NOT %IX1.5.27 AND NOT %IX1.5.29 AND NOT %IX1.5.31 AND NOT %IX2.1.9 AND NOT %IX2.1.13 AND NOT %IX2.1.25 AND NOT %IX2.1.29 AND NOT %IX2.9.1) AND NOT %QX1.4.25 AND NOT %QX1.4.26 THEN
    %ML3600.10 := TRUE;
END_IF;
(* 팝업 메시지 *)
(* Rung L176 *)
IF NOT (NOT %QX1.4.25 AND NOT %QX1.4.26) THEN %ML3600.10 := FALSE; END_IF;
(* Rung L177 *)
IF NOT (NOT %IX1.5.19 AND NOT %IX1.5.23 AND NOT %ML3020.7 AND NOT %ML3020.12 AND NOT %IX1.5.3 AND NOT %IX1.5.7 AND NOT %ML3010.22 AND NOT %ML3010.27 AND NOT %IX1.5.25 AND NOT %IX1.5.27 AND NOT %IX1.5.29 AND NOT %IX1.5.31 AND NOT %IX2.1.9 AND NOT %IX2.1.13 AND NOT %IX2.1.25 AND NOT %IX2.1.29 AND NOT %IX2.9.1) AND NOT %ML202.0 AND NOT %ML202.1 AND NOT %ML202.2 AND NOT %ML202.3 AND NOT %ML202.6 AND NOT %ML202.7 AND NOT %ML202.8 AND NOT %ML202.9 THEN
    %ML3600.11 := TRUE;
END_IF;
(* Rung L178 *)
IF NOT (NOT %ML202.0 AND NOT %ML202.1 AND NOT %ML202.2 AND NOT %ML202.3 AND NOT %ML202.6 AND NOT %ML202.7 AND NOT %ML202.8 AND NOT %ML202.9) THEN
    %ML3600.11 := FALSE;
END_IF;

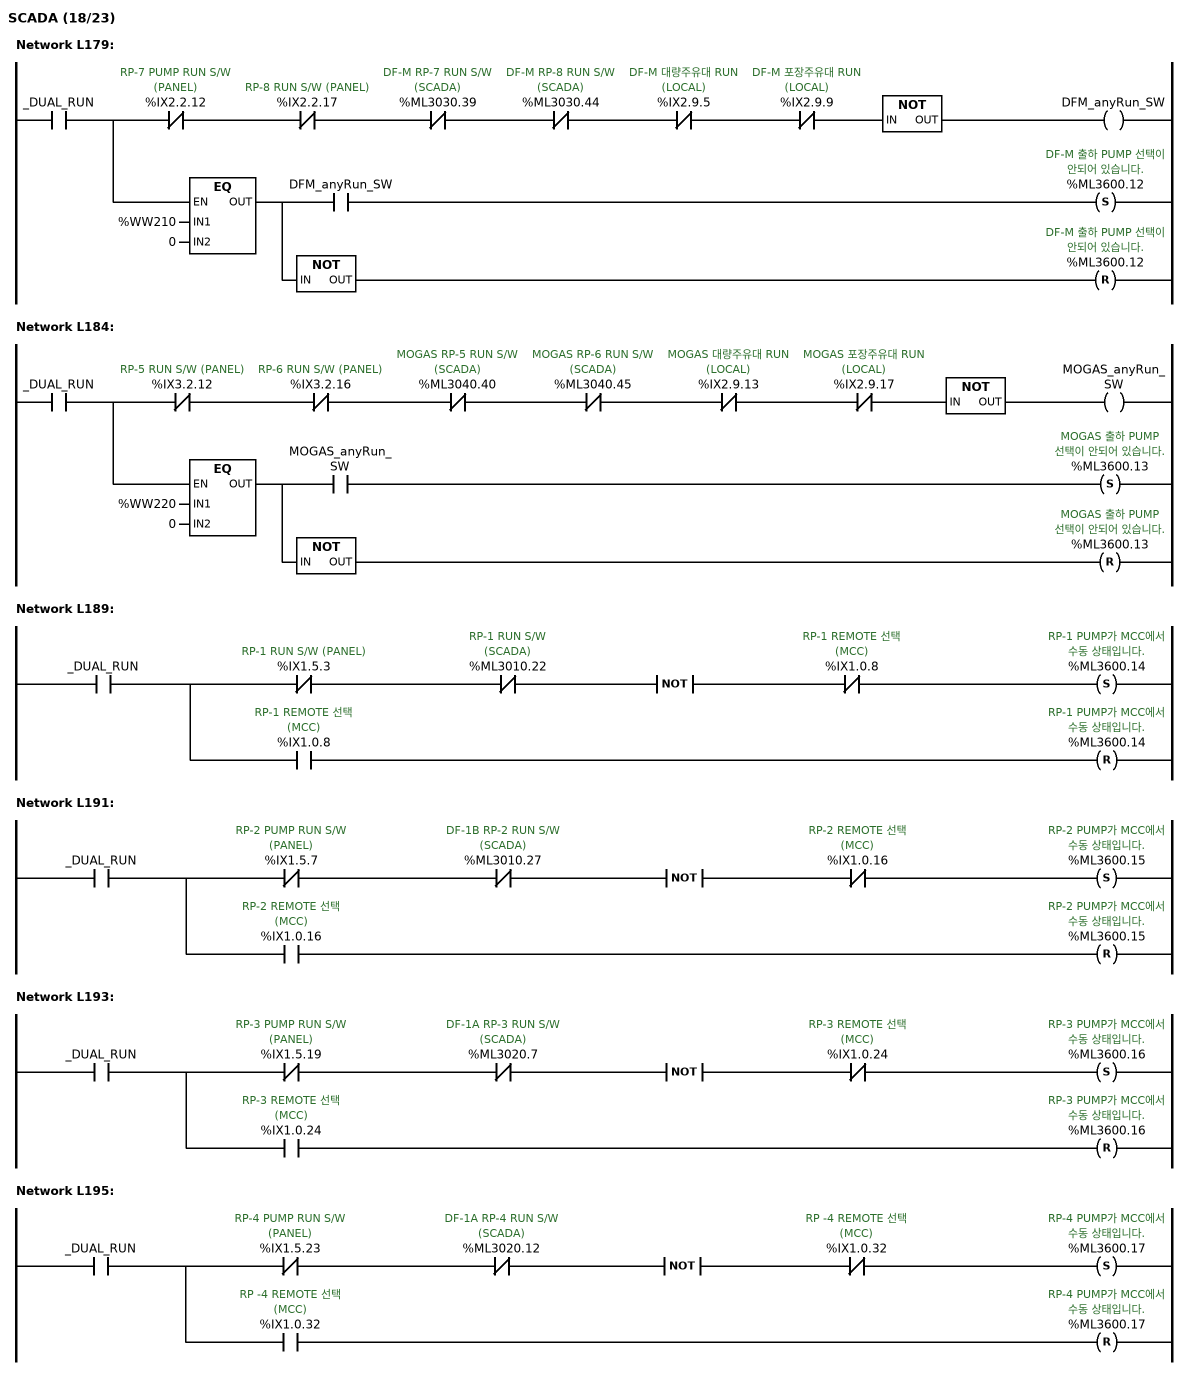
(* Rung L179 *)
DFM_anyRun_SW := NOT (_DUAL_RUN AND NOT %IX2.2.12 AND NOT %IX2.2.17 AND NOT %ML3030.39 AND NOT %ML3030.44 AND NOT %IX2.9.5 AND NOT %IX2.9.9);
IF _DUAL_RUN THEN _t1 := %WW210 = 0; END_IF;
IF _t1 AND DFM_anyRun_SW THEN %ML3600.12 := TRUE; END_IF;
IF NOT _t1 THEN %ML3600.12 := FALSE; END_IF;
(* Rung L184 *)
MOGAS_anyRun_SW := NOT (_DUAL_RUN AND NOT %IX3.2.12 AND NOT %IX3.2.16 AND NOT %ML3040.40 AND NOT %ML3040.45 AND NOT %IX2.9.13 AND NOT %IX2.9.17);
IF _DUAL_RUN THEN _t2 := %WW220 = 0; END_IF;
IF _t2 AND MOGAS_anyRun_SW THEN %ML3600.13 := TRUE; END_IF;
IF NOT _t2 THEN %ML3600.13 := FALSE; END_IF;
(* Rung L189 *)
IF NOT (_DUAL_RUN AND NOT %IX1.5.3 AND NOT %ML3010.22) AND NOT %IX1.0.8 THEN %ML3600.14 := TRUE; END_IF;
IF _DUAL_RUN AND %IX1.0.8 THEN %ML3600.14 := FALSE; END_IF;
(* Rung L191 *)
IF NOT (_DUAL_RUN AND NOT %IX1.5.7 AND NOT %ML3010.27) AND NOT %IX1.0.16 THEN %ML3600.15 := TRUE; END_IF;
IF _DUAL_RUN AND %IX1.0.16 THEN %ML3600.15 := FALSE; END_IF;
(* Rung L193 *)
IF NOT (_DUAL_RUN AND NOT %IX1.5.19 AND NOT %ML3020.7) AND NOT %IX1.0.24 THEN %ML3600.16 := TRUE; END_IF;
IF _DUAL_RUN AND %IX1.0.24 THEN %ML3600.16 := FALSE; END_IF;
(* Rung L195 *)
IF NOT (_DUAL_RUN AND NOT %IX1.5.23 AND NOT %ML3020.12) AND NOT %IX1.0.32 THEN %ML3600.17 := TRUE; END_IF;
IF _DUAL_RUN AND %IX1.0.32 THEN %ML3600.17 := FALSE; END_IF;

